TYPE ACMethodBaseR :
STRUCT
END_STRUCT
END_TYPE

(* stored: Version 1.1.0.1, ProductVersion 3.1.4020.12
   DUT ACMethodBaseR: Id {a0ad6e64-1c56-4c33-83a8-5b53c0554f5b} *)
